Staubli VAL3: start.pgx

program start()
begin

  // call SameInstruct()

  call TestSetmoveid()

end
